// TIA Portal V20 export
// export: Created 2025-12-01T14:56:09.1201688Z, ExportSetting None, DisplayName Totally Integrated Automation Portal, DisplayVersion V20 Update 3, DisplayName TIA Portal Openness, DisplayVersion V20 Update 3, DisplayName TIA Portal Version Control Interface, DisplayVersion V20 Update 3, DisplayName STEP 7 Professional, DisplayVersion V20 Update 3, DisplayName STEP 7 Safety, DisplayVersion V20 Update 2, DisplayName WinCC Basic/Comfort/Advanced, DisplayVersion V20 Update 3, DisplayName WinCC Professional, DisplayVersion V20 Update 3, DisplayName WinCC Unified, DisplayVersion V20 Update 3
TYPE "UDT_EntrePLCs"
   STRUCT
      Mckey : UDInt;
      MesaDestino : UInt;   // Mesa Destino de la UT >>> RUTA[1]
      MesaSiguienteRuta : UInt;   // Mesa Siguiente >>> RUTA[0]
      Grupo : UInt;   // Numero de Grupo de la UT
      TipoCarga : USInt;   // Tipo de Carga
      AtributosDelaCarga : Struct
         Vacia : Bool;   // Atributos Especiales del la Carga --> Vacia
         Pila : Bool;   // Atributos Especiales del la Carga --> Pila
         Remontada : Bool;   // Atributos Especiales del la Carga --> Remontada
      END_STRUCT;
   END_STRUCT;
END_TYPE
